{attribute 'pack_mode' := '1'}

//{attribute 'hide_all_locals'}
TYPE ST_SupervisorHeader :
	STRUCT
		Protocol_version : UINT;
		Message_ID		 : UINT;
		Message_length	 : UDINT;
	END_STRUCT
END_TYPE

//When sending a message from Supervisor to Navitrol, this is populated using F_SetHeaderInfo.

(* stored: Version 1.1.0.1
   DUT ST_SupervisorHeader: Id {77264308-66a8-4f31-8b94-b1e1812d84ee} *)
